{attribute 'GeneratedUsingTerminal: AX8206-0100-0101-0101'}
{attribute addProperty BoxType "AX8206-0100-0101-0101"}
{attribute addProperty Id "Ch_B_AxisMain_InputsCh_B_AxisMain_Inputs_A10B23CB8Ch_B_AxisMain_OutputsCh_B_AxisMain_Outputs_526A47F82Ch_B_Interpolator_OutputsCh_B_Interpolator_Outputs_F819AE728Ch_B_PositionControl_InputsCh_B_PositionControl_Inputs_C884000A4"}
{attribute addProperty CRC "1577601962"}
{attribute addProperty Size "22"}
TYPE Ch_B_5E084BAA :
STRUCT
	{attribute addProperty Name "Ch_B_AxisMain_Inputs"}
	Ch_B_AxisMain_Inputs  : Ch_B_AxisMain_Inputs_A10B23CB;
	{attribute addProperty Name "Ch_B_AxisMain_Outputs"}
	Ch_B_AxisMain_Outputs  : Ch_B_AxisMain_Outputs_526A47F8;
	{attribute addProperty Name "Ch_B_Interpolator_Outputs"}
	Ch_B_Interpolator_Outputs  : Ch_B_Interpolator_Outputs_F819AE72;
	{attribute addProperty Name "Ch_B_PositionControl_Inputs"}
	Ch_B_PositionControl_Inputs  : Ch_B_PositionControl_Inputs_C884000A;
END_STRUCT
END_TYPE

(* stored: Version 1.2.0.0, ProductVersion 3.1.4024.9
   DUT Ch_B_5E084BAA: Id {3778d48a-7365-407f-b4b1-ffff90f30c15} *)
